SYSTEM Kulbana System
  (* Version 1.0, 2005-06-13, Goran, Chalmers *)
  DEVICE Test Device : DeviceType_not_used
    RESOURCE TestResource : ResourceType_not_used
      FBS
        restart : E_RESTART;
        merge2 : E_MERGE2;
        splitStor : E_SPLIT2;
        splitLiten : E_SPLIT2;
        kulbana : Kulbana;
        matlyft : KulaMatlyft;
        matstation : Matstation;
        hiss : Hiss;
        van1 : Kullager;
        van2 : Kullager;
        arm : Arm;
      END_FBS
      EVENT_CONNECTIONS
        restart.COLD TO kulbana.INIT;
        kulbana.INITO TO merge2.EI1;
        merge2.EO TO kulbana.InPortvakt;
        kulbana.KulaPortvakt TO kulbana.UrPortvakt;
        kulbana.KulaMatlyft TO matlyft.KulaMatlyft;
        kulbana.MatlyftNere TO matlyft.MatlyftNere;
        matlyft.UppMatlyft TO kulbana.UppMatlyft;
        kulbana.StorKula TO splitStor.EI;
        kulbana.LitenKula TO splitLiten.EI;
        kulbana.KulaMatstation TO matstation.KulaMatstation;
        splitStor.EO1 TO matstation.Storkula;
        splitLiten.EO1 TO matstation.Litenkula;
        matstation.Mat TO kulbana.Mat;
        matstation.Urmatning TO kulbana.UrMatning;
        splitStor.EO2 TO hiss.StorKula;
        splitLiten.EO2 TO hiss.LitenKula;
        kulbana.KulaHiss TO hiss.KulaHiss;
        kulbana.HissNere TO hiss.HissNere;
        hiss.UppHissVan1 TO kulbana.UppHissVan1;
        hiss.UppHissVan2 TO kulbana.UppHissVan2;
        kulbana.KulaVan1 TO van1.KULAFRAMME;
        van1.PUTTAUT TO kulbana.UtVan1;
        kulbana.KulaVan2 TO van2.KULAFRAMME;
        van2.PUTTAUT TO kulbana.UtVan2;
        kulbana.PlockaVan1 TO arm.PlockaVan1;
        kulbana.PlockaVan2 TO arm.PlockaVan2;
        kulbana.ArmVan1 TO arm.ArmVan1;
        kulbana.ArmVan2 TO arm.ArmVan2;
        arm.UppArmVan1 TO kulbana.UppArmVan1;
        arm.UppArmVan2 TO kulbana.UppArmVan2;
        arm.ArmHem TO kulbana.ArmHem;
        kulbana.ArmHemma TO merge2.EI2;
      END_CONNECTIONS
    END_RESOURCE
  END_DEVICE
END_SYSTEM
